{attribute 'qualified_only'}
VAR_GLOBAL PERSISTENT
	user_array 					: ARRAY[1..100] OF ST_UserManagment;  // Tablica użytkowników
    currentUser 				: INT := 1;  // Indeks bieżącego użytkownika (zaczyna od 1)
	outside_login_pool			:STRING(255);  
	currentUserName 			:WSTRING(255);
	currentUserGroup			:STRING(80);
	currentUserGroupNumber		:UINT;
	putted_user_password		:STRING(255);  //pole w które użytkownik wpisuje hasło
	newuserNameSurname 			:WSTRING(255);	//imię i nazwisko
	newpassword					:STRING(255);	//hasło
	newpasswordRFID				:STRING(255);	//hasło rfid
	newpasswordQR				:STRING(255);	//hasło qr
	newuserGroup				:STRING(80);		//grupa użytkowników
	newuserGroupNumber			:UINT;
	newautoLogOff				:STRING(80);			//czas do wylogowania
	actual_editted_user			:WSTRING(255);	//wybór aktualnie edytowanego użytkownika
	edituserNameSurname 		:WSTRING(255);	//imię i nazwisko
	editpassword				:STRING(255);	//hasło
	editpasswordRFID			:STRING(255);	//hasło rfid
	editpasswordQR				:STRING(255);	//hasło qr
	edituserGroup				:STRING(80);	//grupa użytkowników
	editUserGroupNumber			:UINT;
	editautoLogOff				:STRING(80);	//czas do wylogowania


END_VAR
VAR_GLOBAL
	new_user_add_error			:BOOL;
	edit_user_error				:BOOL;
	bwait						:BOOL;
	delete_user					:BOOL;
	delete_user_accept			:BOOL;
	delete_user_error			:BOOL;
	choosen_to_delete			:WSTRING(255);
	user_deleted_succes			:BOOL;
	password_to_log_in			:STRING(80); //hasło do pola (1 z 5 (adm, opr, ser, tech, mech	
	b_rewrite_users_after_issues:BOOL:=FALSE;
	b_user_drop_the_login		:BOOL;
	i_choosen_language 			:INT:=1;
	outside_accept_login		:BOOL;
	logout						:BOOL;
	user_try_to_log				:BOOL;
	user_accept_to_log_in		:BOOL;
	no_user_found				:BOOL;
	user_succesed_log			:BOOL;
	edit_user_qr_or_rfid_password :BOOL;		//edycja kodów rfid lub qr
	new_user_added				:BOOL;		//dodano użytkownika w PLC
	user_eddited				:BOOL; 		//zedytowano użytkownika w PLC
	b_new_users					:BOOL;		//wgranie uzytkowników
	new_user					:BOOL;			//inicjalizacja dodawania nowego użytkownika
	new_user_accept				:BOOL;			//akceptacja dodania nowego użytkownika
	edit_user					:BOOL;				//inicjalizacja edycji użytkownika
	edit_user_accept			:BOOL;			//akceptacja edycji użytkownika
	actualUserOn_UserName		:STRING(80);
	b_rewrite_main_users		:BOOL:=FALSE;
	string_of_properties 		: STRING(1000);  // String z HMI z danymi użytkowników
END_VAR

(* stored: Version 1.1.0.1, ProductVersion 3.1.4026.13, FileIdentifier 1a75394454372ed0782eb6e2fcd698312981b287, FileSignature 455dfa76c22786fb369748bb12ce9fd5dc656e7c682639aa449134a4d060e565353bce5dfd64be21a7174859dae7f9b83aed87a653d56e9990ac190c0c425ef516458380447205d32a35ea0a20bf1ea4dcc121fab35afb5218f21ebb3d6c65de89dd25e354a57534e6ac7b62d59f9ac98ca27f88faac98916ab56112c962ff11c9af1bff6507435c3bfd5b711e9d3bedf54262a9b6401b4784c45f234fe52fbb9a27c6906597e465f923734d9e6e3e7b84f2b127ceb6caf006a3c11da9c05e2ccc674f1931090873f0ccbbb696505f8c454d2d1240eb2ecc5653d1e7cd0e55c6b4e40acdce30896a4cbed9b2001204a66b631dc6de2100bd7a53d074f98d52f2
   GVL GVL_USER: Id {286f2749-1eaf-4ba8-975d-c30c224cc4fb} *)
